KUKA KRL data list: ps_b_etb_res_c02.dat

&ACCESS RVO1
&COMMENT Solda Axor ETB
&PARAM DISKPATH = KRC:\R1\Program\OLP
DEFDAT ps_b_etb_res_c02
;FOLD EXTERNAL DECLARATIONS;%{PE}%MKUKATPBASIS,%CEXT,%VCOMMON,%P
;FOLD GRIPPERTECH EXT
EXT  H50 (INT  :IN,INT  :IN,INT  :IN,GRP_TYP  :IN )
;ENDFOLD (GRIPPERTECH EXT)
;FOLD SPOTTECH EXT
EXT  USERSPOT (S_COMMAND  :IN,SPOT_TYPE  :IN )
;ENDFOLD (SPOTTECH EXT)
;FOLD BASISTECH EXT;%{PE}%MKUKATPBASIS,%CEXT,%VEXT,%P
EXT  BAS (BAS_COMMAND  :IN,REAL  :IN )
DECL INT SUCCESS
;ENDFOLD (BASISTECH EXT)
;FOLD USER EXT;%{E}%MKUKATPUSER,%CEXT,%VEXT,%P
;Make your modifications here

;ENDFOLD (USER EXT)
;ENDFOLD (EXTERNAL DECLARATIONS)


DECL FDAT Fl035={TOOL_NO 3,BASE_NO 3,IPO_FRAME #BASE,POINT2[] " "}
DECL E6POS Xl035={X 584.140991,Y 789.36499,Z 1229.97498,A 158.485001,B 12.9363003,C 166.735794,S 2,T 42}
DECL LDAT LL_OLP8={VEL 2.0,ACC 100.0,APO_DIST 0.0,APO_FAC 0.0,ORI_TYP #VAR,CIRC_TYP #BASE,JERK_FAC 50.0}
DECL FDAT Fl040={TOOL_NO 3,BASE_NO 3,IPO_FRAME #BASE,POINT2[] " "}
DECL E6POS Xl040={X 565.49762,Y 693.462708,Z 1207.63196,A 154.968201,B 9.37270164,C 157.367493,S 18,T 42,E1 0.0,E2 0.0,E3 0.0,E4 0.0,E5 0.0,E6 0.0}
DECL LDAT LL_OLP9={VEL 2.0,ACC 100.0,APO_DIST 0.0,APO_FAC 0.0,ORI_TYP #VAR,CIRC_TYP #BASE,JERK_FAC 50.0}


DECL FDAT Fl045={TOOL_NO 3,BASE_NO 3,IPO_FRAME #BASE,POINT2[] " "}
DECL E6POS Xl045={X 561.989014,Y 691.565002,Z 1096.26794,A 154.969498,B 9.37310028,C 147.3685,S 2,T 42}



DECL LDAT LL_OLP10={VEL 2.0,ACC 100.0,APO_DIST 0.0,APO_FAC 0.0,ORI_TYP #VAR,CIRC_TYP #BASE,JERK_FAC 50.0}





DECL FDAT Fl060={TOOL_NO 3,BASE_NO 3,IPO_FRAME #BASE,POINT2[] " "}
DECL E6POS Xl060={X 618.291992,Y 968.916992,Z 1209.96594,A -149.936798,B -80.7937012,C 61.0236015,S 2,T 34}
DECL LDAT LL_OLP13={VEL 2.0,ACC 100.0,APO_DIST 0.0,APO_FAC 0.0,ORI_TYP #VAR,CIRC_TYP #BASE,JERK_FAC 50.0}
DECL FDAT Fl065={TOOL_NO 3,BASE_NO 3,IPO_FRAME #BASE,POINT2[] " "}
DECL E6POS Xl065={X 584.655212,Y 961.50769,Z 1277.37,A -132.780594,B -83.9849777,C 40.2847786,S 18,T 34,E1 0.0,E2 0.0,E3 0.0,E4 0.0,E5 0.0,E6 0.0}
DECL LDAT LL_OLP14={VEL 2.0,ACC 100.0,APO_DIST 0.0,APO_FAC 0.0,ORI_TYP #VAR,CIRC_TYP #BASE,JERK_FAC 50.0}
DECL FDAT FSWP_60_7788={TOOL_NO 3,BASE_NO 3,IPO_FRAME #BASE,POINT2[] " "}
DECL E6POS XSWP_60_7788={X 593.953918,Y 986.767883,Z 1318.20398,A -158.466003,B -86.9588623,C 65.2502365,S 18,T 34,E1 0.0,E2 0.0,E3 0.0,E4 0.0,E5 0.0,E6 0.0}
DECL LDAT LL_OLP15={VEL 2.0,ACC 100.0,APO_DIST 0.0,APO_FAC 0.0,ORI_TYP #VAR,CIRC_TYP #BASE,JERK_FAC 50.0}
DECL FDAT FSWP_60_7790={TOOL_NO 3,BASE_NO 3,IPO_FRAME #BASE,POINT2[] " ",TQ_STATE FALSE}
DECL E6POS XSWP_60_7790={X 630.814392,Y 987.352783,Z 1320.06995,A 140.791306,B -87.3468628,C 128.899902,S 18,T 34,E1 0.0,E2 0.0,E3 0.0,E4 0.0,E5 0.0,E6 0.0}
DECL LDAT LL_OLP16={VEL 2.0,ACC 100.0,APO_DIST 0.0,APO_FAC 0.0,ORI_TYP #VAR,CIRC_TYP #BASE,JERK_FAC 50.0}
DECL FDAT FSWP_60_7792={TOOL_NO 3,BASE_NO 3,IPO_FRAME #BASE,POINT2[] " "}
DECL E6POS XSWP_60_7792={X 662.207397,Y 986.047485,Z 1321.43396,A 149.066498,B -87.567482,C 121.761398,S 18,T 34,E1 0.0,E2 0.0,E3 0.0,E4 0.0,E5 0.0,E6 0.0}
DECL LDAT LL_OLP17={VEL 2.0,ACC 100.0,APO_DIST 0.0,APO_FAC 0.0,ORI_TYP #VAR,CIRC_TYP #BASE,JERK_FAC 50.0}










DECL FDAT FSWP_60_7796={TOOL_NO 3,BASE_NO 3,IPO_FRAME #BASE,POINT2[] " "}
DECL E6POS XSWP_60_7796={X 732.090088,Y 986.195129,Z 1321.95703,A 8.9285593,B -75.0170364,C -96.2651367,S 18,T 34,E1 0.0,E2 0.0,E3 0.0,E4 0.0,E5 0.0,E6 0.0}
DECL LDAT LL_OLP22={VEL 2.0,ACC 100.0,APO_DIST 0.0,APO_FAC 0.0,ORI_TYP #VAR,CIRC_TYP #BASE,JERK_FAC 50.0}
DECL FDAT FSWP_60_7798={TOOL_NO 3,BASE_NO 3,IPO_FRAME #BASE,POINT2[] " "}
DECL E6POS XSWP_60_7798={X 776.076782,Y 986.822021,Z 1321.77197,A 4.67742491,B -75.0973969,C -92.1623077,S 18,T 34,E1 0.0,E2 0.0,E3 0.0,E4 0.0,E5 0.0,E6 0.0}
DECL LDAT LL_OLP23={VEL 2.0,ACC 100.0,APO_DIST 0.0,APO_FAC 0.0,ORI_TYP #VAR,CIRC_TYP #BASE,JERK_FAC 50.0}
DECL FDAT FSWP_60_7800={TOOL_NO 3,BASE_NO 3,IPO_FRAME #BASE,POINT2[] " "}
DECL E6POS XSWP_60_7800={X 823.064087,Y 986.974182,Z 1321.75305,A 4.2844758,B -75.2971115,C -91.1988983,S 18,T 34,E1 0.0,E2 0.0,E3 0.0,E4 0.0,E5 0.0,E6 0.0}
DECL LDAT LL_OLP24={VEL 2.0,ACC 100.0,APO_DIST 0.0,APO_FAC 0.0,ORI_TYP #VAR,CIRC_TYP #BASE,JERK_FAC 50.0}
DECL FDAT FSWP_60_7802={TOOL_NO 3,BASE_NO 3,IPO_FRAME #BASE,POINT2[] " "}
DECL E6POS XSWP_60_7802={X 868.485474,Y 987.476807,Z 1322.875,A -7.07572317,B -75.2149582,C -79.7813568,S 18,T 34,E1 0.0,E2 0.0,E3 0.0,E4 0.0,E5 0.0,E6 0.0}
DECL LDAT LL_OLP25={VEL 2.0,ACC 100.0,APO_DIST 0.0,APO_FAC 0.0,ORI_TYP #VAR,CIRC_TYP #BASE,JERK_FAC 50.0}
DECL FDAT FSWP_60_7804={TOOL_NO 3,BASE_NO 3,IPO_FRAME #BASE,POINT2[] " "}
DECL E6POS XSWP_60_7804={X 914.553772,Y 988.416626,Z 1322.60498,A -5.14426804,B -75.1808929,C -81.9923935,S 18,T 34,E1 0.0,E2 0.0,E3 0.0,E4 0.0,E5 0.0,E6 0.0}
DECL LDAT LL_OLP26={VEL 2.0,ACC 100.0,APO_DIST 0.0,APO_FAC 0.0,ORI_TYP #VAR,CIRC_TYP #BASE,JERK_FAC 50.0}
DECL FDAT FSWP_60_7808={TOOL_NO 3,BASE_NO 3,IPO_FRAME #BASE,POINT2[] " "}
DECL E6POS XSWP_60_7808={X 1012.69897,Y 988.867493,Z 1321.68103,A -9.06076431,B -74.9903564,C -78.263031,S 18,T 34,E1 0.0,E2 0.0,E3 0.0,E4 0.0,E5 0.0,E6 0.0}
DECL LDAT LL_OLP27={VEL 2.0,ACC 100.0,APO_DIST 0.0,APO_FAC 0.0,ORI_TYP #VAR,CIRC_TYP #BASE,JERK_FAC 50.0}
DECL FDAT FSWP_60_7810={TOOL_NO 3,BASE_NO 3,IPO_FRAME #BASE,POINT2[] " "}
DECL E6POS XSWP_60_7810={X 1060.17603,Y 988.960815,Z 1322.047,A -9.69721889,B -74.9386597,C -77.70224,S 18,T 34,E1 0.0,E2 0.0,E3 0.0,E4 0.0,E5 0.0,E6 0.0}
DECL LDAT LL_OLP28={VEL 2.0,ACC 100.0,APO_DIST 0.0,APO_FAC 0.0,ORI_TYP #VAR,CIRC_TYP #BASE,JERK_FAC 50.0}
DECL FDAT FSWP_60_7812={TOOL_NO 3,BASE_NO 3,IPO_FRAME #BASE,POINT2[] " "}
DECL E6POS XSWP_60_7812={X 1103.52502,Y 989.145874,Z 1321.01501,A -11.5189104,B -74.7814102,C -76.1083527,S 18,T 34,E1 0.0,E2 0.0,E3 0.0,E4 0.0,E5 0.0,E6 0.0}
DECL LDAT LL_OLP29={VEL 2.0,ACC 100.0,APO_DIST 0.0,APO_FAC 0.0,ORI_TYP #VAR,CIRC_TYP #BASE,JERK_FAC 50.0}
DECL FDAT FSWP_60_7814={TOOL_NO 3,BASE_NO 3,IPO_FRAME #BASE,POINT2[] " "}
DECL E6POS XSWP_60_7814={X 1147.04895,Y 989.444214,Z 1319.48499,A -9.90039444,B -74.9102325,C -77.5600281,S 18,T 34,E1 0.0,E2 0.0,E3 0.0,E4 0.0,E5 0.0,E6 0.0}
DECL LDAT LL_OLP30={VEL 2.0,ACC 100.0,APO_DIST 0.0,APO_FAC 0.0,ORI_TYP #VAR,CIRC_TYP #BASE,JERK_FAC 50.0}
DECL FDAT FSWP_60_7816={TOOL_NO 3,BASE_NO 3,IPO_FRAME #BASE,POINT2[] " "}
DECL E6POS XSWP_60_7816={X 1193.93994,Y 989.052429,Z 1318.43799,A -3.23020291,B -75.0366669,C -84.5184631,S 18,T 34,E1 0.0,E2 0.0,E3 0.0,E4 0.0,E5 0.0,E6 0.0}
DECL LDAT LL_OLP31={VEL 2.0,ACC 100.0,APO_DIST 0.0,APO_FAC 0.0,ORI_TYP #VAR,CIRC_TYP #BASE,JERK_FAC 50.0}
DECL FDAT Fl090={TOOL_NO 3,BASE_NO 3,IPO_FRAME #BASE,POINT2[] " "}
DECL E6POS Xl090={X 1197.92505,Y 977.659119,Z 1291.51294,A -14.5019197,B -74.4627228,C -73.6420135,S 18,T 34,E1 0.0,E2 0.0,E3 0.0,E4 0.0,E5 0.0,E6 0.0}
DECL LDAT LL_OLP32={VEL 2.0,ACC 100.0,APO_DIST 0.0,APO_FAC 0.0,ORI_TYP #VAR,CIRC_TYP #BASE,JERK_FAC 50.0}
DECL FDAT Fl095={TOOL_NO 3,BASE_NO 3,IPO_FRAME #BASE,POINT2[] " "}
DECL E6POS Xl095={X 1176.72498,Y 986.589111,Z 1209.34399,A -44.4494286,B -83.9011688,C -44.0611382,S 18,T 34,E1 0.0,E2 0.0,E3 0.0,E4 0.0,E5 0.0,E6 0.0}
















DECL FDAT Fl120={TOOL_NO 3,BASE_NO 3,IPO_FRAME #BASE,POINT2[] " "}

DECL E6POS Xl120={X 1303.89905,Y 1020.01202,Z 107.1138,A 179.976105,B -22.3131905,C 89.996582,S 18,T 34,E1 0.0,E2 0.0,E3 0.0,E4 0.0,E5 0.0,E6 0.0}
DECL LDAT LL_OLP38={VEL 2.0,ACC 100.0,APO_DIST 0.0,APO_FAC 0.0,ORI_TYP #VAR,CIRC_TYP #BASE,JERK_FAC 50.0}

DECL FDAT FSWP_60_7488={TOOL_NO 3,BASE_NO 3,IPO_FRAME #BASE,POINT2[] " "}

DECL E6POS XSWP_60_7488={X 1311.22095,Y 1033.19299,Z 111.022697,A 179.772202,B -22.2714005,C 89.0542221,S 18,T 34,E1 0.0,E2 0.0,E3 0.0,E4 0.0,E5 0.0,E6 0.0}
DECL LDAT LL_OLP39={VEL 2.0,ACC 100.0,APO_DIST 0.0,APO_FAC 0.0,ORI_TYP #VAR,CIRC_TYP #BASE,JERK_FAC 50.0}

DECL FDAT FSWP_60_7490={TOOL_NO 3,BASE_NO 3,IPO_FRAME #BASE,POINT2[] " "}

DECL E6POS XSWP_60_7490={X 1343.11304,Y 1034.01001,Z 112.712502,A 179.979401,B -22.3128395,C 90.9136963,S 18,T 34,E1 0.0,E2 0.0,E3 0.0,E4 0.0,E5 0.0,E6 0.0}
DECL LDAT LL_OLP40={VEL 2.0,ACC 100.0,APO_DIST 0.0,APO_FAC 0.0,ORI_TYP #VAR,CIRC_TYP #BASE,JERK_FAC 50.0}

DECL FDAT FSWP_60_7492={TOOL_NO 3,BASE_NO 3,IPO_FRAME #BASE,POINT2[] " "}

DECL E6POS XSWP_60_7492={X 1374.13794,Y 1032.24304,Z 112.369598,A 179.975098,B -22.3114605,C 90.5738602,S 18,T 34,E1 0.0,E2 0.0,E3 0.0,E4 0.0,E5 0.0,E6 0.0}
DECL LDAT LL_OLP41={VEL 2.0,ACC 100.0,APO_DIST 0.0,APO_FAC 0.0,ORI_TYP #VAR,CIRC_TYP #BASE,JERK_FAC 50.0}

DECL FDAT Fl125={TOOL_NO 3,BASE_NO 3,IPO_FRAME #BASE,POINT2[] " "}


DECL E6POS Xl125={X 1397.44604,Y 1024.76294,Z 95.6467438,A 179.9758,B -17.5534992,C 89.9962769,S 18,T 34,E1 0.0,E2 0.0,E3 0.0,E4 0.0,E5 0.0,E6 0.0}
DECL LDAT LL_OLP42={VEL 2.0,ACC 100.0,APO_DIST 0.0,APO_FAC 0.0,ORI_TYP #VAR,CIRC_TYP #BASE,JERK_FAC 50.0}
DECL FDAT Fl130={TOOL_NO 3,BASE_NO 3,IPO_FRAME #BASE,POINT2[] " "}
DECL E6POS Xl130={X 1469.67896,Y 1023.99103,Z 98.598999,A 179.975601,B -17.0133991,C 89.9968033,S 2,T 34}
DECL LDAT LL_OLP43={VEL 2.0,ACC 100.0,APO_DIST 0.0,APO_FAC 0.0,ORI_TYP #VAR,CIRC_TYP #BASE,JERK_FAC 50.0}



DECL FDAT FSWP_60_7496={TOOL_NO 3,BASE_NO 3,IPO_FRAME #BASE,POINT2[] " "}

DECL E6POS XSWP_60_7496={X 1451.93506,Y 1031.19397,Z 116.244598,A 179.984207,B -21.8104496,C 94.6474533,S 18,T 42,E1 0.0,E2 0.0,E3 0.0,E4 0.0,E5 0.0,E6 0.0}
DECL LDAT LL_OLP44={VEL 2.0,ACC 100.0,APO_DIST 0.0,APO_FAC 0.0,ORI_TYP #VAR,CIRC_TYP #BASE,JERK_FAC 50.0}

DECL FDAT FSWP_60_7498={TOOL_NO 3,BASE_NO 3,IPO_FRAME #BASE,POINT2[] " "}


DECL E6POS XSWP_60_7498={X 1491.30701,Y 1029.375,Z 115.388397,A -179.990005,B -23.6027298,C 93.9890137,S 18,T 34,E1 0.0,E2 0.0,E3 0.0,E4 0.0,E5 0.0,E6 0.0}
DECL LDAT LL_OLP45={VEL 2.0,ACC 100.0,APO_DIST 0.0,APO_FAC 0.0,ORI_TYP #VAR,CIRC_TYP #BASE,JERK_FAC 50.0}
DECL FDAT FSWP_60_7500={TOOL_NO 3,BASE_NO 3,IPO_FRAME #BASE,POINT2[] " "}
DECL E6POS XSWP_60_7500={X 1535.73303,Y 1028.76501,Z 113.8647,A -179.940399,B -26.5961704,C 93.7221298,S 18,T 34,E1 0.0,E2 0.0,E3 0.0,E4 0.0,E5 0.0,E6 0.0}
DECL LDAT LL_OLP46={VEL 2.0,ACC 100.0,APO_DIST 0.0,APO_FAC 0.0,ORI_TYP #VAR,CIRC_TYP #BASE,JERK_FAC 50.0}

DECL FDAT Fl140={TOOL_NO 3,BASE_NO 3,IPO_FRAME #BASE,POINT2[] " "}
DECL PDAT PP_OLP2={VEL 100.0,ACC 100.0,APO_DIST 0.0,APO_MODE #CDIS}
DECL E6POS Xl140={X 1610.60205,Y 1139.57495,Z 45.987999,A 179.975998,B -22.3132992,C 89.9968033,S 2,T 34}
DECL BASIS_SUGG_T LAST_BASIS={POINT1[] "P0                      ",POINT2[] "P0                      ",CP_PARAMS[] "CPDAT0                  ",PTP_PARAMS[] "PDAT0                   ",CONT[] "                        ",CP_VEL[] "2.0                     ",PTP_VEL[] " 100                    ",SYNC_PARAMS[] "SYNCDAT                 ",SPL_NAME[] "S0                      "}
DECL PDAT PP_OLP4={VEL 100.0,ACC 100.0,APO_DIST 30.0,APO_MODE #CDIS}
DECL E6POS Xl006={X 1083.797,Y 1451.30701,Z 836.236023,A 174.173294,B -30.1965008,C 118.184799,S 2,T 42}
DECL FDAT Fl006={TOOL_NO 3,BASE_NO 3,IPO_FRAME #BASE,POINT2[] " "}
DECL LDAT LL_OLP48={VEL 2.0,ACC 100.0,APO_DIST 30.0,APO_FAC 0.0,ORI_TYP #VAR,CIRC_TYP #BASE,JERK_FAC 50.0}
DECL E6POS Xl011={X 563.752014,Y 1566.71301,Z 1132.11096,A 154.969406,B 9.37310028,C 157.3685,S 2,T 42}
DECL FDAT Fl011={TOOL_NO 3,BASE_NO 3,IPO_FRAME #BASE,POINT2[] " "}
DECL LDAT LL_OLP49={VEL 2.0,ACC 100.0,APO_DIST 0.0,APO_FAC 0.0,ORI_TYP #VAR,CIRC_TYP #BASE,JERK_FAC 50.0}
DECL E6POS Xl016={X 563.297913,Y 691.402771,Z 1151.29895,A 154.970306,B 9.36947632,C 147.371796,S 18,T 42,E1 0.0,E2 0.0,E3 0.0,E4 0.0,E5 0.0,E6 0.0}
DECL FDAT Fl016={TOOL_NO 3,BASE_NO 3,IPO_FRAME #BASE,POINT2[] " "}
DECL PDAT PP_OLP5={VEL 100.0,ACC 100.0,APO_DIST 0.0}
DECL E6POS Xl021={X 564.475891,Y 693.618713,Z 1160.99097,A 154.970398,B 9.36874485,C 157.370407,S 18,T 42,E1 0.0,E2 0.0,E3 0.0,E4 0.0,E5 0.0,E6 0.0}
DECL FDAT Fl021={TOOL_NO 3,BASE_NO 3,IPO_FRAME #BASE,POINT2[] " "}
DECL LDAT LL_OLP50={VEL 2.0,ACC 100.0,APO_DIST 30.0,APO_FAC 0.0,ORI_TYP #VAR,CIRC_TYP #BASE,JERK_FAC 50.0}
DECL E6POS Xl026={X 299.222107,Y 607.531128,Z 1021.26202,A 157.030594,B 37.3611107,C 158.838806,S 18,T 42,E1 0.0,E2 0.0,E3 0.0,E4 0.0,E5 0.0,E6 0.0}
DECL FDAT Fl026={TOOL_NO 3,BASE_NO 3,IPO_FRAME #BASE,POINT2[] " "}












DECL LDAT LL_OLP51={VEL 2.0,ACC 100.0,APO_DIST 0.0,APO_FAC 0.0,ORI_TYP #VAR,CIRC_TYP #BASE,JERK_FAC 50.0}
DECL E6POS Xl031={X 99.1301804,Y 417.839813,Z 796.104614,A 160.762802,B 75.7358627,C 165.230301,S 18,T 42,E1 0.0,E2 0.0,E3 0.0,E4 0.0,E5 0.0,E6 0.0}
DECL FDAT Fl031={TOOL_NO 3,BASE_NO 3,IPO_FRAME #BASE,POINT2[] " "}
DECL PDAT PP_OLP6={VEL 100.0,ACC 100.0,APO_DIST 0.0}
DECL E6POS Xl036={X 100.0737,Y 399.872711,Z 769.99469,A 161.946793,B 77.1953964,C 165.6996,S 18,T 42,E1 0.0,E2 0.0,E3 0.0,E4 0.0,E5 0.0,E6 0.0}
DECL FDAT Fl036={TOOL_NO 3,BASE_NO 3,IPO_FRAME #BASE,POINT2[] " "}
DECL PDAT PP_OLP7={VEL 100.0,ACC 100.0,APO_DIST 10.0,APO_MODE #CDIS}
DECL E6POS Xl041={X 104.556396,Y 364.301605,Z 731.724792,A 164.799805,B 79.9908905,C 167.122696,S 18,T 42,E1 0.0,E2 0.0,E3 0.0,E4 0.0,E5 0.0,E6 0.0}
DECL FDAT Fl041={TOOL_NO 3,BASE_NO 3,IPO_FRAME #BASE,POINT2[] " "}
DECL LDAT LL_OLP52={VEL 2.0,ACC 100.0,APO_DIST 0.0,APO_FAC 0.0,ORI_TYP #VAR,CIRC_TYP #BASE,JERK_FAC 50.0}
DECL E6POS Xl046={X 91.8286896,Y 379.290894,Z 653.815796,A 159.358994,B 82.8835907,C 161.735306,S 18,T 42,E1 0.0,E2 0.0,E3 0.0,E4 0.0,E5 0.0,E6 0.0}
DECL FDAT Fl046={TOOL_NO 3,BASE_NO 3,IPO_FRAME #BASE,POINT2[] " "}
DECL LDAT LL_OLP53={VEL 2.0,ACC 100.0,APO_DIST 0.0,APO_FAC 0.0,ORI_TYP #VAR,CIRC_TYP #BASE,JERK_FAC 50.0}
DECL E6POS XSWP_60_9280={X 95.6109619,Y 381.409088,Z 613.008728,A 154.631805,B 84.2475128,C 156.982895,S 18,T 42,E1 0.0,E2 0.0,E3 0.0,E4 0.0,E5 0.0,E6 0.0}
DECL FDAT FSWP_60_9280={TOOL_NO 3,BASE_NO 3,IPO_FRAME #BASE,POINT2[] " "}
DECL LDAT LL_OLP54={VEL 2.0,ACC 100.0,APO_DIST 0.0,APO_FAC 0.0,ORI_TYP #VAR,CIRC_TYP #BASE,JERK_FAC 50.0}
DECL E6POS XSWP_60_9282={X 96.4919968,Y 412.008606,Z 612.211304,A 160.145096,B 82.8769302,C 161.574799,S 18,T 42,E1 0.0,E2 0.0,E3 0.0,E4 0.0,E5 0.0,E6 0.0}
DECL FDAT FSWP_60_9282={TOOL_NO 3,BASE_NO 3,IPO_FRAME #BASE,POINT2[] " "}
DECL LDAT LL_OLP55={VEL 2.0,ACC 100.0,APO_DIST 0.0,APO_FAC 0.0,ORI_TYP #VAR,CIRC_TYP #BASE,JERK_FAC 50.0}
DECL E6POS XSWP_60_9286={X 98.8377228,Y 478.136993,Z 615.090515,A 158.5354,B 82.6687012,C 159.334305,S 18,T 42,E1 0.0,E2 0.0,E3 0.0,E4 0.0,E5 0.0,E6 0.0}
DECL FDAT FSWP_60_9286={TOOL_NO 3,BASE_NO 3,IPO_FRAME #BASE,POINT2[] " "}
DECL LDAT LL_OLP56={VEL 2.0,ACC 100.0,APO_DIST 0.0,APO_FAC 0.0,ORI_TYP #VAR,CIRC_TYP #BASE,JERK_FAC 50.0}
DECL E6POS XSWP_60_9288={X 103.058403,Y 513.388794,Z 616.070129,A 159.082199,B 82.9015808,C 159.794006,S 18,T 42,E1 0.0,E2 0.0,E3 0.0,E4 0.0,E5 0.0,E6 0.0}
DECL FDAT FSWP_60_9288={TOOL_NO 3,BASE_NO 3,IPO_FRAME #BASE,POINT2[] " "}
DECL LDAT LL_OLP57={VEL 2.0,ACC 100.0,APO_DIST 0.0,APO_FAC 0.0,ORI_TYP #VAR,CIRC_TYP #BASE,JERK_FAC 50.0}
DECL E6POS XSWP_60_9290={X 104.816704,Y 545.921387,Z 613.990295,A 160.234207,B 82.8796921,C 161.131805,S 18,T 42,E1 0.0,E2 0.0,E3 0.0,E4 0.0,E5 0.0,E6 0.0}
DECL FDAT FSWP_60_9290={TOOL_NO 3,BASE_NO 3,IPO_FRAME #BASE,POINT2[] " "}
DECL LDAT LL_OLP58={VEL 2.0,ACC 100.0,APO_DIST 0.0,APO_FAC 0.0,ORI_TYP #VAR,CIRC_TYP #BASE,JERK_FAC 50.0}
DECL E6POS XSWP_60_9292={X 106.351799,Y 574.419678,Z 615.045471,A 159.705002,B 82.8796616,C 161.683899,S 18,T 42,E1 0.0,E2 0.0,E3 0.0,E4 0.0,E5 0.0,E6 0.0}
DECL FDAT FSWP_60_9292={TOOL_NO 3,BASE_NO 3,IPO_FRAME #BASE,POINT2[] " "}
DECL LDAT LL_OLP59={VEL 2.0,ACC 100.0,APO_DIST 0.0,APO_FAC 0.0,ORI_TYP #VAR,CIRC_TYP #BASE,JERK_FAC 50.0}
DECL E6POS XSWP_60_9296={X 111.656799,Y 646.356079,Z 614.34491,A 159.402298,B 82.8827896,C 161.777603,S 18,T 42,E1 0.0,E2 0.0,E3 0.0,E4 0.0,E5 0.0,E6 0.0}
DECL FDAT FSWP_60_9296={TOOL_NO 3,BASE_NO 3,IPO_FRAME #BASE,POINT2[] " "}
DECL LDAT LL_OLP60={VEL 2.0,ACC 100.0,APO_DIST 0.0,APO_FAC 0.0,ORI_TYP #VAR,CIRC_TYP #BASE,JERK_FAC 50.0}
DECL E6POS XSWP_60_9298={X 114.739799,Y 682.679688,Z 615.256714,A 159.398407,B 82.8830185,C 161.775497,S 18,T 42,E1 0.0,E2 0.0,E3 0.0,E4 0.0,E5 0.0,E6 0.0}
DECL FDAT FSWP_60_9298={TOOL_NO 3,BASE_NO 3,IPO_FRAME #BASE,POINT2[] " "}
DECL LDAT LL_OLP61={VEL 2.0,ACC 100.0,APO_DIST 0.0,APO_FAC 0.0,ORI_TYP #VAR,CIRC_TYP #BASE,JERK_FAC 50.0}
DECL E6POS XSWP_60_9300={X 118.410202,Y 718.615112,Z 616.465881,A 159.434296,B 82.8800735,C 161.813599,S 18,T 42,E1 0.0,E2 0.0,E3 0.0,E4 0.0,E5 0.0,E6 0.0}
DECL FDAT FSWP_60_9300={TOOL_NO 3,BASE_NO 3,IPO_FRAME #BASE,POINT2[] " "}
DECL LDAT LL_OLP62={VEL 2.0,ACC 100.0,APO_DIST 0.0,APO_FAC 0.0,ORI_TYP #VAR,CIRC_TYP #BASE,JERK_FAC 50.0}
DECL E6POS XSWP_60_9302={X 121.885803,Y 754.708618,Z 617.715881,A 159.414902,B 82.8859329,C 161.790604,S 18,T 42,E1 0.0,E2 0.0,E3 0.0,E4 0.0,E5 0.0,E6 0.0}
DECL FDAT FSWP_60_9302={TOOL_NO 3,BASE_NO 3,IPO_FRAME #BASE,POINT2[] " "}
DECL LDAT LL_OLP63={VEL 2.0,ACC 100.0,APO_DIST 0.0,APO_FAC 0.0,ORI_TYP #VAR,CIRC_TYP #BASE,JERK_FAC 50.0}
DECL E6POS XSWP_60_9304={X 127.169601,Y 790.217773,Z 618.741577,A 159.411896,B 82.8858337,C 161.788101,S 18,T 42,E1 0.0,E2 0.0,E3 0.0,E4 0.0,E5 0.0,E6 0.0}
DECL FDAT FSWP_60_9304={TOOL_NO 3,BASE_NO 3,IPO_FRAME #BASE,POINT2[] " "}
DECL LDAT LL_OLP64={VEL 2.0,ACC 100.0,APO_DIST 0.0,APO_FAC 0.0,ORI_TYP #VAR,CIRC_TYP #BASE,JERK_FAC 50.0}
DECL E6POS XSWP_60_9306={X 135.140793,Y 844.331726,Z 621.312012,A 159.393005,B 82.8853378,C 161.772095,S 18,T 42,E1 0.0,E2 0.0,E3 0.0,E4 0.0,E5 0.0,E6 0.0}
DECL FDAT FSWP_60_9306={TOOL_NO 3,BASE_NO 3,IPO_FRAME #BASE,POINT2[] " "}
DECL LDAT LL_OLP65={VEL 2.0,ACC 100.0,APO_DIST 0.0,APO_FAC 0.0,ORI_TYP #VAR,CIRC_TYP #BASE,JERK_FAC 50.0}
DECL E6POS XSWP_60_9322={X 142.100906,Y 879.108521,Z 618.917114,A 159.403595,B 82.8969116,C 167.300201,S 18,T 42,E1 0.0,E2 0.0,E3 0.0,E4 0.0,E5 0.0,E6 0.0}
DECL FDAT FSWP_60_9322={TOOL_NO 3,BASE_NO 3,IPO_FRAME #BASE,POINT2[] " "}
DECL E6POS Xl051={X 137.945007,Y 854.049988,Z 676.479004,A 164.794098,B 79.9898987,C 167.113907,S 2,T 42}
DECL FDAT Fl051={TOOL_NO 3,BASE_NO 3,IPO_FRAME #BASE,POINT2[] " "}
DECL SPOT_TYPE SNORMAL={GUN 1,PAIR #FIRST,RETR #OPN,CLO_TM 0,PGNO1 1,PRESS1 0.0,PGNO2 0,PRESS2 0.0}
DECL E6POS XP3={X 254.703003,Y 563.97522,Z 963.619019,A 158.715103,B 51.3612404,C 160.321594,S 18,T 42,E1 0.0,E2 0.0,E3 0.0,E4 0.0,E5 0.0,E6 0.0}
DECL FDAT FP3={TOOL_NO 3,BASE_NO 3,IPO_FRAME #BASE,POINT2[] " ",TQ_STATE FALSE}
DECL LDAT LCPDAT2={VEL 2.0,ACC 100.0,APO_DIST 10.0,APO_FAC 50.0,AXIS_VEL 100.0,AXIS_ACC 100.0,ORI_TYP #VAR,CIRC_TYP #BASE,JERK_FAC 50.0,GEAR_JERK 50.0,EXAX_IGN 0}
DECL E6POS XP6={X 96.662323,Y 417.583801,Z 818.442078,A 160.817001,B 73.6449432,C 162.906403,S 18,T 42,E1 0.0,E2 0.0,E3 0.0,E4 0.0,E5 0.0,E6 0.0}
DECL FDAT FP6={TOOL_NO 3,BASE_NO 3,IPO_FRAME #BASE,POINT2[] " ",TQ_STATE FALSE}
DECL LDAT LCPDAT5={VEL 2.0,ACC 100.0,APO_DIST 100.0,APO_FAC 50.0,AXIS_VEL 100.0,AXIS_ACC 100.0,ORI_TYP #VAR,CIRC_TYP #BASE,JERK_FAC 50.0,GEAR_JERK 50.0,EXAX_IGN 0}
DECL E6POS XP7={X 151.468903,Y 490.672791,Z 892.769409,A 160.394699,B 62.3519096,C 161.4758,S 18,T 42,E1 0.0,E2 0.0,E3 0.0,E4 0.0,E5 0.0,E6 0.0}
DECL FDAT FP7={TOOL_NO 3,BASE_NO 3,IPO_FRAME #BASE,POINT2[] " ",TQ_STATE FALSE}
DECL LDAT LCPDAT6={VEL 2.0,ACC 100.0,APO_DIST 100.0,APO_FAC 50.0,AXIS_VEL 100.0,AXIS_ACC 100.0,ORI_TYP #VAR,CIRC_TYP #BASE,JERK_FAC 50.0,GEAR_JERK 50.0,EXAX_IGN 0}
DECL E6POS XP8={X 98.0387115,Y 417.105408,Z 795.282715,A 160.479095,B 75.2753067,C 164.7733,S 18,T 42,E1 0.0,E2 0.0,E3 0.0,E4 0.0,E5 0.0,E6 0.0}
DECL FDAT FP8={TOOL_NO 3,BASE_NO 3,IPO_FRAME #BASE,POINT2[] " ",TQ_STATE FALSE}
DECL LDAT LCPDAT7={VEL 2.0,ACC 100.0,APO_DIST 100.0,APO_FAC 50.0,AXIS_VEL 100.0,AXIS_ACC 100.0,ORI_TYP #VAR,CIRC_TYP #BASE,JERK_FAC 50.0,GEAR_JERK 50.0,EXAX_IGN 0}


DECL E6POS XP11={X 1560.58704,Y 1009.72302,Z 65.5483475,A 179.964401,B -43.8393517,C 90.9567795,S 18,T 34,E1 0.0,E2 0.0,E3 0.0,E4 0.0,E5 0.0,E6 0.0}
DECL FDAT FP11={TOOL_NO 3,BASE_NO 3,IPO_FRAME #BASE,POINT2[] " ",TQ_STATE FALSE}

DECL LDAT LCPDAT10={VEL 2.0,ACC 100.0,APO_DIST 100.0,APO_FAC 50.0,AXIS_VEL 100.0,AXIS_ACC 100.0,ORI_TYP #VAR,CIRC_TYP #BASE,JERK_FAC 50.0,GEAR_JERK 50.0,EXAX_IGN 0}
DECL SPOT_SUGG_T LAST_SPOT={GUN[] "1                       ",RETR_CMD[] "#OPN                    ",CHOISE[] "#FIRST                  ",CLO_TM[] "0                       ",PGNO1[] "1                       ",PRESS1[] "0                       ",PGNO2[] "1                       ",PRESS2[] "0                       ",SPOT_PARAMS[] "NORMAL                  "}
DECL E6POS XP14={X 1610.68799,Y 1340.54297,Z 45.7100296,A 179.967102,B -22.3057804,C 90.001152,S 18,T 34,E1 0.0,E2 0.0,E3 0.0,E4 0.0,E5 0.0,E6 0.0}
DECL FDAT FP14={TOOL_NO 3,BASE_NO 3,IPO_FRAME #BASE,POINT2[] " ",TQ_STATE FALSE}
DECL PDAT PPDAT5={VEL 100.0,ACC 95.0,APO_DIST 100.0,APO_MODE #CDIS,GEAR_JERK 50.0}
DECL E6POS XP16={X 1711.52502,Y 2023.51099,Z 556.947876,A -175.166397,B -41.1158485,C 86.8608398,S 18,T 34,E1 0.0,E2 0.0,E3 0.0,E4 0.0,E5 0.0,E6 0.0}
DECL FDAT FP16={TOOL_NO 3,BASE_NO 3,IPO_FRAME #BASE,POINT2[] " ",TQ_STATE FALSE}
DECL PDAT PPDAT7={VEL 100.0,ACC 100.0,APO_DIST 100.0,APO_MODE #CDIS,GEAR_JERK 50.0}
DECL E6POS XP17={X 1711.651,Y 2023.50098,Z 556.917297,A -175.160202,B -41.1122093,C 86.8591003,S 18,T 42,E1 0.0,E2 0.0,E3 0.0,E4 0.0,E5 0.0,E6 0.0}


DECL FDAT FP17={TOOL_NO 3,BASE_NO 3,IPO_FRAME #BASE,POINT2[] " ",TQ_STATE FALSE}
DECL PDAT PPDAT8={VEL 100.0,ACC 100.0,APO_DIST 100.0,APO_MODE #CDIS,GEAR_JERK 50.0}
DECL LDAT LCPDAT11={VEL 2.0,ACC 100.0,APO_DIST 10.0,APO_FAC 50.0,AXIS_VEL 100.0,AXIS_ACC 100.0,ORI_TYP #VAR,CIRC_TYP #BASE,JERK_FAC 50.0,GEAR_JERK 50.0,EXAX_IGN 0}
DECL E6POS XP18={X 60.9463196,Y 487.706207,Z 619.175598,A 160.159195,B 82.8793716,C 161.610504,S 18,T 42,E1 0.0,E2 0.0,E3 0.0,E4 0.0,E5 0.0,E6 0.0}
DECL FDAT FP18={TOOL_NO 3,BASE_NO 3,IPO_FRAME #BASE,POINT2[] " ",TQ_STATE FALSE}
DECL LDAT LCPDAT12={VEL 2.0,ACC 100.0,APO_DIST 10.0,APO_FAC 50.0,AXIS_VEL 100.0,AXIS_ACC 100.0,ORI_TYP #VAR,CIRC_TYP #BASE,JERK_FAC 50.0,GEAR_JERK 50.0,EXAX_IGN 0}

DECL E6POS XP19={X 128.315308,Y 824.686523,Z 636.831726,A 156.575699,B 83.7855835,C 158.972504,S 18,T 42,E1 0.0,E2 0.0,E3 0.0,E4 0.0,E5 0.0,E6 0.0}

DECL FDAT FP19={TOOL_NO 3,BASE_NO 3,IPO_FRAME #BASE,POINT2[] " ",TQ_STATE FALSE}

DECL LDAT LL_OLP68={VEL 2.0,ACC 100.0,APO_DIST 10.0,APO_FAC 0.0,ORI_TYP #VAR,CIRC_TYP #BASE,JERK_FAC 50.0}
DECL E6POS Xl037={X 416.389008,Y 806.565979,Z 1106.76904,A 158.978607,B 33.3137093,C 165.382401,S 18,T 42,E1 0.0,E2 0.0,E3 0.0,E4 0.0,E5 0.0,E6 0.0}
DECL FDAT Fl037={TOOL_NO 3,BASE_NO 3,IPO_FRAME #BASE,POINT2[] " "}


DECL LDAT LL_OLP69={VEL 2.0,ACC 100.0,APO_DIST 0.0,APO_FAC 0.0,ORI_TYP #VAR,CIRC_TYP #BASE,JERK_FAC 50.0}
DECL E6POS XSWP_60_9258={X 150.526398,Y 915.172119,Z 620.970825,A 92.024292,B 54.5307693,C 101.880798,S 18,T 42,E1 0.0,E2 0.0,E3 0.0,E4 0.0,E5 0.0,E6 0.0}
DECL FDAT FSWP_60_9258={TOOL_NO 3,BASE_NO 3,IPO_FRAME #BASE,POINT2[] " ",TQ_STATE FALSE}
DECL LDAT LCPDAT15={VEL 2.0,ACC 100.0,APO_DIST 5.0,APO_FAC 50.0,AXIS_VEL 100.0,AXIS_ACC 100.0,ORI_TYP #VAR,CIRC_TYP #BASE,JERK_FAC 50.0,GEAR_JERK 50.0,EXAX_IGN 0}
DECL LDAT LCPDAT16={VEL 2.0,ACC 100.0,APO_DIST 0.0,APO_FAC 50.0,AXIS_VEL 100.0,AXIS_ACC 100.0,ORI_TYP #VAR,CIRC_TYP #BASE,JERK_FAC 50.0,GEAR_JERK 50.0,EXAX_IGN 0}
DECL LDAT LCPDAT0={VEL 2.0,ACC 100.0,APO_DIST 30.0,APO_FAC 50.0,AXIS_VEL 100.0,AXIS_ACC 100.0,ORI_TYP #VAR,CIRC_TYP #BASE,JERK_FAC 50.0,GEAR_JERK 50.0,EXAX_IGN 0}
DECL E6POS Xl066={X 1312.10205,Y 1148.0,Z 79.7080002,A 180.0,B -13.3133001,C 90.0,S 2,T 42}
DECL FDAT Fl066={TOOL_NO 3,BASE_NO 3,IPO_FRAME #BASE,POINT2[] " "}
DECL LDAT LCPDAT17={VEL 2.0,ACC 100.0,APO_DIST 5.0,APO_FAC 50.0,AXIS_VEL 100.0,AXIS_ACC 100.0,ORI_TYP #VAR,CIRC_TYP #BASE,JERK_FAC 50.0,GEAR_JERK 50.0,EXAX_IGN 0}
DECL E6POS XP22={X 1230.61096,Y 1015.41901,Z 62.1031799,A -179.999207,B -13.3151903,C 90.0011368,S 18,T 42,E1 0.0,E2 0.0,E3 0.0,E4 0.0,E5 0.0,E6 0.0}
DECL FDAT FP22={TOOL_NO 3,BASE_NO 3,IPO_FRAME #BASE,POINT2[] " ",TQ_STATE FALSE}
DECL LDAT LL_OLP70={VEL 2.0,ACC 100.0,APO_DIST 5.0,APO_FAC 0.0,ORI_TYP #VAR,CIRC_TYP #BASE,JERK_FAC 50.0}
DECL E6POS Xl071={X 1116.63403,Y 1017.16602,Z 51.4317093,A 179.996597,B -13.3109398,C 90.0032806,S 18,T 42,E1 0.0,E2 0.0,E3 0.0,E4 0.0,E5 0.0,E6 0.0}
DECL FDAT Fl071={TOOL_NO 3,BASE_NO 3,IPO_FRAME #BASE,POINT2[] " ",TQ_STATE FALSE}
DECL LDAT LCPDAT18={VEL 2.0,ACC 100.0,APO_DIST 5.0,APO_FAC 50.0,AXIS_VEL 100.0,AXIS_ACC 100.0,ORI_TYP #VAR,CIRC_TYP #BASE,JERK_FAC 50.0,GEAR_JERK 50.0,EXAX_IGN 0}
DECL E6POS XP23={X 1108.78296,Y 1017.35999,Z 73.2284927,A 179.996597,B -13.3102198,C 90.0024872,S 18,T 42,E1 0.0,E2 0.0,E3 0.0,E4 0.0,E5 0.0,E6 0.0}
DECL FDAT FP23={TOOL_NO 3,BASE_NO 3,IPO_FRAME #BASE,POINT2[] " ",TQ_STATE FALSE}
DECL LDAT LCPDAT19={VEL 2.0,ACC 100.0,APO_DIST 100.0,APO_FAC 50.0,AXIS_VEL 100.0,AXIS_ACC 100.0,ORI_TYP #VAR,CIRC_TYP #BASE,JERK_FAC 50.0,GEAR_JERK 50.0,EXAX_IGN 0}
DECL E6POS XSWP_61_7028={X 1106.74695,Y 1027.08203,Z 71.4262695,A 179.0914,B -13.2747402,C 90.0131607,S 18,T 42,E1 0.0,E2 0.0,E3 0.0,E4 0.0,E5 0.0,E6 0.0}
DECL FDAT FSWP_61_7028={TOOL_NO 3,BASE_NO 3,IPO_FRAME #BASE,POINT2[] " ",TQ_STATE FALSE}
DECL LDAT LCPDAT20={VEL 2.0,ACC 100.0,APO_DIST 100.0,APO_FAC 50.0,AXIS_VEL 100.0,AXIS_ACC 100.0,ORI_TYP #VAR,CIRC_TYP #BASE,JERK_FAC 50.0,GEAR_JERK 50.0,EXAX_IGN 0}
DECL E6POS XSWP_61_7030={X 1150.88794,Y 1030.36304,Z 88.9034576,A -179.999802,B -13.3076496,C 90.0065002,S 18,T 42,E1 0.0,E2 0.0,E3 0.0,E4 0.0,E5 0.0,E6 0.0}
DECL FDAT FSWP_61_7030={TOOL_NO 3,BASE_NO 3,IPO_FRAME #BASE,POINT2[] " ",TQ_STATE FALSE}
DECL LDAT LCPDAT21={VEL 2.0,ACC 100.0,APO_DIST 100.0,APO_FAC 50.0,AXIS_VEL 100.0,AXIS_ACC 100.0,ORI_TYP #VAR,CIRC_TYP #BASE,JERK_FAC 50.0,GEAR_JERK 50.0,EXAX_IGN 0}
DECL E6POS XSWP_61_7032={X 1219.53101,Y 1034.36597,Z 101.103302,A -179.906494,B -19.7676105,C 90.0269394,S 18,T 34,E1 0.0,E2 0.0,E3 0.0,E4 0.0,E5 0.0,E6 0.0}
DECL FDAT FSWP_61_7032={TOOL_NO 3,BASE_NO 3,IPO_FRAME #BASE,POINT2[] " ",TQ_STATE FALSE}
DECL LDAT LCPDAT22={VEL 2.0,ACC 100.0,APO_DIST 10.0,APO_FAC 50.0,AXIS_VEL 100.0,AXIS_ACC 100.0,ORI_TYP #VAR,CIRC_TYP #BASE,JERK_FAC 50.0,GEAR_JERK 50.0,EXAX_IGN 0}
DECL E6POS XP24={X 1206.38403,Y 1006.83502,Z 67.4408493,A -179.908997,B -19.7681408,C 90.0280304,S 18,T 34,E1 0.0,E2 0.0,E3 0.0,E4 0.0,E5 0.0,E6 0.0}
DECL FDAT FP24={TOOL_NO 3,BASE_NO 3,IPO_FRAME #BASE,POINT2[] " ",TQ_STATE FALSE}
DECL LDAT LCPDAT23={VEL 2.0,ACC 100.0,APO_DIST 10.0,APO_FAC 50.0,AXIS_VEL 100.0,AXIS_ACC 100.0,ORI_TYP #VAR,CIRC_TYP #BASE,JERK_FAC 50.0,GEAR_JERK 50.0,EXAX_IGN 0}
DECL E6POS XP25={X 1318.55103,Y 1023.52502,Z 83.9089737,A 179.978394,B -22.2589493,C 89.9975967,S 18,T 34,E1 0.0,E2 0.0,E3 0.0,E4 0.0,E5 0.0,E6 0.0}
DECL FDAT FP25={TOOL_NO 3,BASE_NO 3,IPO_FRAME #BASE,POINT2[] " ",TQ_STATE FALSE}
DECL LDAT LL_OLP71={VEL 2.0,ACC 100.0,APO_DIST 0.0,APO_FAC 0.0,ORI_TYP #VAR,CIRC_TYP #BASE,JERK_FAC 50.0}
DECL E6POS Xl052={X 563.752014,Y 1566.71301,Z 1132.11096,A 154.969406,B 9.37310028,C 157.3685,S 2,T 42}
DECL FDAT Fl052={TOOL_NO 3,BASE_NO 3,IPO_FRAME #BASE,POINT2[] " "}
DECL LDAT LL_OLP72={VEL 2.0,ACC 100.0,APO_DIST 0.0,APO_FAC 0.0,ORI_TYP #VAR,CIRC_TYP #BASE,JERK_FAC 50.0}
DECL E6POS Xl056={X 878.794006,Y 1301.91504,Z 1209.96802,A -149.936798,B -80.7937012,C 61.0237007,S 2,T 34}
DECL FDAT Fl056={TOOL_NO 3,BASE_NO 3,IPO_FRAME #BASE,POINT2[] " "}
DECL LDAT LL_OLP73={VEL 2.0,ACC 100.0,APO_DIST 10.0,APO_FAC 0.0,ORI_TYP #VAR,CIRC_TYP #BASE,JERK_FAC 50.0}
DECL E6POS Xl101={X 795.249023,Y 1246.63,Z 1059.69897,A -149.936401,B -80.7937012,C 61.023201,S 2,T 34}
DECL FDAT Fl101={TOOL_NO 3,BASE_NO 3,IPO_FRAME #BASE,POINT2[] " "}
DECL LDAT LL_OLP74={VEL 2.0,ACC 100.0,APO_DIST 30.0,APO_FAC 0.0,ORI_TYP #VAR,CIRC_TYP #BASE,JERK_FAC 50.0}
DECL E6POS Xl106={X 1304.23706,Y 1333.34302,Z 23.5721092,A -179.994904,B -25.5595093,C 89.9953537,S 18,T 34,E1 0.0,E2 0.0,E3 0.0,E4 0.0,E5 0.0,E6 0.0}
DECL FDAT Fl106={TOOL_NO 3,BASE_NO 3,IPO_FRAME #BASE,POINT2[] " "}
DECL PDAT PPDAT1={VEL 100.0,ACC 100.0,APO_DIST 0.0,APO_MODE #CDIS,GEAR_JERK 50.0}
ENDDAT
